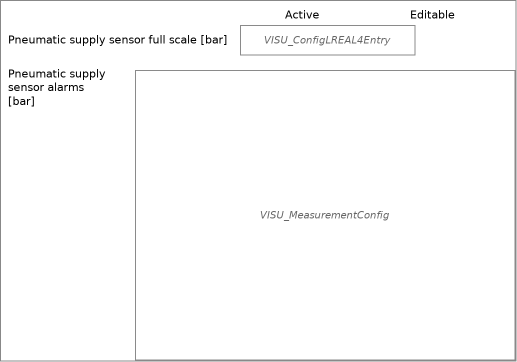
VISUALIZATION VISU_M1Config_General  // 517x362
VAR_IN_OUT
    editable : M1Config;
	active : M1Config;
END_VAR
    Label (240,5 125x20), "Active"
    Label (370,5 125x20), "Editable"
    Label (5,25 235x30), "Pneumatic supply sensor full scale [bar]"
    Frame (240,25 175x30)
        shows VISU_ConfigLREAL4Entry(active := active.pneumaticSupplySensorFullScale, editable := editable.pneumaticSupplySensorFullScale)
    Label (5,60 105x55), "Pneumatic supply sensor alarms [bar]"
    Frame (135,70 380x290)
        shows VISU_MeasurementConfig(active := active.pneumaticSupplyPressure, editable := editable.pneumaticSupplyPressure)
END_VISUALIZATION

(* stored: Version 1.1.0.1, ProductVersion 3.1.4019.2
   Visu VISU_M1Config_General: Id {e970b92b-667c-40fa-a053-b7c2b81e01fa} *)
